// Creates a Sift Proxy Protocol "create_ingestion_config" Endpoint Message.
FUNCTION _F_CreateIngestionConfigMessage 

VAR_INPUT
	stIngestionConfig : REFERENCE TO ST_IngestionConfig;
	stMsg : REFERENCE TO _ST_SiftMessage;
	pJsonBuffer : POINTER TO BYTE;
	nLength : UDINT;
END_VAR

VAR
	fbJson : FB_JsonSaxWriter;
	i : UDINT;
	j : UDINT;
	k : UDINT;
	tmpChannelConfig : REFERENCE TO ST_ChannelConfig;
	tmpEnumType : REFERENCE TO ST_EnumType;
	pJsonString : POINTER TO STRING;
	nBytes : UDINT;
END_VAR

VAR_OUTPUT
	stErr : ST_SiftError;
END_VAR

IF pJsonBuffer = 0 THEN
	stErr.bError := TRUE;
	stErr.nErrId := GVL_SIFT.NULL_JSON_POINTER;
	stErr.sReason := 'The JSON buffer is null';
	RETURN;
END_IF

fbJson.StartObject();

fbJson.AddKey('asset_name');
fbJson.AddString(stIngestionConfig.sAssetName);

fbJson.AddKey('flows');
fbJson.StartArray();
FOR i := 1 TO stIngestionConfig.nNumFlowConfigs DO
	fbJson.StartObject();

	fbJson.AddKey('name');
	fbJson.AddString(stIngestionConfig.aFlowConfigs[i-1].sName);

	fbJson.AddKey('channels');
	fbJson.StartArray();
	FOR j := 1 TO stIngestionConfig.aFlowConfigs[i-1].nNumChannelConfigs DO
		fbJson.StartObject();
		tmpChannelConfig REF= stIngestionConfig.aFlowConfigs[i-1].aChannelConfigs[j-1];

		fbJson.AddKey('name');
		fbJson.AddString(tmpChannelConfig.sName);

		IF tmpChannelConfig.sUnit <> '' THEN
			fbJson.AddKey('unit');
			fbJson.AddString(tmpChannelConfig.sUnit);
		END_IF
		
		IF tmpChannelConfig.sDescription <> '' THEN
			fbJson.AddKey('description');
			fbJson.AddString(tmpChannelConfig.sDescription);
		END_IF
	
		fbJson.AddKey('data_type');
		CASE tmpChannelConfig.eDataType OF
			E_ChannelDataType.Bool_:
				fbJson.AddString('CHANNEL_DATA_TYPE_BOOL');
			
			E_ChannelDataType.Double:
				fbJson.AddString('CHANNEL_DATA_TYPE_DOUBLE');
			
			E_ChannelDataType.Enum:
				fbJson.AddString('CHANNEL_DATA_TYPE_ENUM');
			
			E_ChannelDataType.Float:
				fbJson.AddString('CHANNEL_DATA_TYPE_FLOAT');
			
			E_ChannelDataType.Int32:
				fbJson.AddString('CHANNEL_DATA_TYPE_INT_32');
			
			E_ChannelDataType.Int64:
				fbJson.AddString('CHANNEL_DATA_TYPE_INT_64');
			
			E_ChannelDataType.String_:
				fbJson.AddString('CHANNEL_DATA_TYPE_STRING');
			
			E_ChannelDataType.Uint32:
				fbJson.AddString('CHANNEL_DATA_TYPE_UINT_32');

			E_ChannelDataType.Uint64:
				fbJson.AddString('CHANNEL_DATA_TYPE_UINT_64');
		END_CASE
		
		fbJson.AddKey('enum_types');
		fbJson.StartArray();
		FOR k := 1 TO tmpChannelConfig.nNumEnumTypes DO
			tmpEnumType REF= tmpChannelConfig.aEnumTypes[k-1];
			fbJson.StartObject();
			
			fbJson.AddKey('name');
			fbJson.AddString(tmpEnumType.sName);
			
			fbJson.AddKey('key');
			fbJson.AddUdint(tmpEnumType.nKey);
			
			fbJson.EndObject();
		END_FOR
		fbJson.EndArray();
		
		fbJson.EndObject();
	END_FOR
	fbJson.EndArray();
		
	fbJson.EndObject();
END_FOR
fbJson.EndArray();

fbJson.EndObject();

pJsonString := pJsonBuffer;
nBytes := fbJson.CopyDocument(pJsonString^, nLength);
IF nBytes = 0 THEN
	stErr.nErrId := GVL_SIFT.JSON_CAPACITY_REACHED;
	stErr.bError := TRUE;
	stErr.sReason := CONCAT(
		CONCAT('JSON msg too large: ', UDINT_TO_STRING(fbJson.GetDocumentLength())),
		' endpoint=create_ingestion_config',
	);
	RETURN;
END_IF

stErr := _F_CreateEndpointMessage(sEndpoint:='create_ingestion_config', 
                                  pData:=pJsonString, 
                                  nLength:=nBytes-1,
                                  nBufferLength := nLength, 
                                  stMsg:=stMsg);

END_FUNCTION

(* stored: Version 1.1.0.1
   POU _F_CreateIngestionConfigMessage: Id {e5079918-0a05-4adf-bee4-a1d66848a106}, SpecialFunc None *)
